// TwinCAT 3 PLC project home
// ProgramVersion: 3.1.4024.0
// libraries:
//   Tc2_Standard, * (Beckhoff Automation GmbH)
//   Tc2_System, * (Beckhoff Automation GmbH)
//   Tc3_Module, * (Beckhoff Automation GmbH)
// project tree:
//   / Food.TcDUT, Fridge.TcDUT, garden.TcPOU, house.TcGVL, Kitchen.TcPOU, main.TcPOU, Plant.TcDUT, Room.TcPOU, task_garden.TcTTO, task_house.TcTTO
// real-time tasks:
//   TASK task_house: cycle T#10ms, priority 20, ADS port 350
//   TASK task_garden: cycle T#10ms, priority 1, ADS port 351

CONFIGURATION home
    RESOURCE PLC ON TwinCAT3
        TASK task_garden(INTERVAL := T#10ms, PRIORITY := 1);
        TASK task_house(INTERVAL := T#10ms, PRIORITY := 20);
        PROGRAM garden WITH task_garden : garden;
        PROGRAM main WITH task_house : main;
    END_RESOURCE
END_CONFIGURATION

// ---- Food.TcDUT
{attribute 'qualified_only'}
{attribute 'strict'}
{attribute 'to_string'}
TYPE Food :
(
    Nothing,
    Carrot,
    Cabbage,
    Broccoli,
    Peas,
    Tofu,
    Humous,
    LentilCurry
);
END_TYPE

// ---- Fridge.TcDUT
TYPE Fridge :
STRUCT
// Store meat at the bottom
    top_shelf    : ARRAY [0..7] OF Food;
    middle_shelf : ARRAY [0..7] OF Food;
    bottom_shelf : ARRAY [0..7] OF Food;
    drawer       : ARRAY [0..3] OF Food;
    door_shelf   : ARRAY [0..3] OF Food;
END_STRUCT
END_TYPE

// ---- Plant.TcDUT
{attribute 'qualified_only'}
{attribute 'strict'}
TYPE Plant :
(
    AppleTree,
    BlackberryBush,
    Grass,
    Ivy,
    Hedge,
    RoseBush
);
END_TYPE

// ---- house.TcGVL
{attribute 'qualified_only'}
VAR_GLOBAL CONSTANT
    ADDRESS     : STRING := '13 Apple Cart Way'; // Next door to 1 Pear Drop Lane
    N_BEDROOMS  : USINT  := 4;
    N_BATHROOMS : USINT  := 1;
END_VAR

// ---- garden.TcPOU
PROGRAM garden
VAR PERSISTENT
    plants                  : ARRAY [0..255] OF Plant;
END_VAR
VAR
    vegetable_plot_at_front : ARRAY [0..4] OF ARRAY [0..2] OF ARRAY [0..7] OF Plant;
    vegetable_plot_at_back  : ARRAY [0..3,0..5,0..6] OF Plant;
END_VAR

END_PROGRAM

// ---- main.TcPOU
PROGRAM main
VAR
    kitchen     : Kitchen;
    dining_room : Room;
    living_room : Room;
    bedroom     : ARRAY [0..(house.N_BEDROOMS-1)]  OF Room;
    bathroom    : ARRAY [0..(house.N_BATHROOMS-1)] OF Room;

    i           : USINT := 0;
END_VAR

kitchen(target_luminosity_lumens := 1300, target_temperature_oc := 19.5, n_broccolis := 3);
dining_room(target_luminosity_lumens := 1100, target_temperature_oc := 19.5);
living_room(target_luminosity_lumens := 800, target_temperature_oc := 19.5);

FOR i := 0 TO (house.N_BEDROOMS-1) DO
    bedroom[i](target_luminosity_lumens := 600, target_temperature_oc := 16.0);
END_FOR

FOR i := 0 TO (house.N_BATHROOMS-1) DO
    bathroom[i](target_luminosity_lumens := 1300, target_temperature_oc := 18.5);
END_FOR

END_PROGRAM

// ---- Kitchen.TcPOU
FUNCTION_BLOCK kitchen EXTENDS room
VAR_INPUT
    n_broccolis : USINT := 0;
END_VAR
VAR PERSISTENT
    fridge      : Fridge;
END_VAR
VAR
    description : STRING := '';
    i           : USINT  := 0;
END_VAR

FOR i := 0 TO MIN(n_broccolis, 7) DO
    fridge.top_shelf[i] := Food.Broccoli;
END_FOR

fridge.middle_shelf[4] := Food.Humous;
fridge.middle_shelf[5] := Food.Tofu;

fridge.bottom_shelf[2] := Food.LentilCurry;

fridge.drawer[0] := Food.Peas;

fridge.door_shelf[0] := Food.Nothing;
fridge.door_shelf[1] := Food.Nothing;
fridge.door_shelf[2] := Food.Nothing;
fridge.door_shelf[3] := Food.Nothing;

description := TO_STRING(fridge.top_shelf[0]);

END_FUNCTION_BLOCK

// ---- Room.TcPOU
FUNCTION_BLOCK room
VAR_INPUT
    target_luminosity_lumens : UINT := 1000;
    target_temperature_oc    : REAL := 18.5;
END_VAR
VAR PERSISTENT
    name                     : STRING;
END_VAR
VAR
    actual_luminosity_lumens : UINT := 1200;
    actual_temperature_oc    : REAL := 18.5;
    is_occupied              : BOOL := FALSE;
    heating_on               : BOOL := FALSE;
END_VAR

heating_on := heating();

METHOD PRIVATE heating : BOOL
VAR_INST
    heating_on                    : BOOL := FALSE;
    was_occupied_at_previous_step : BOOL := FALSE;
    timer                         : TON;
END_VAR
IF is_occupied THEN
    timer(IN := FALSE);
ELSIF was_occupied_at_previous_step AND NOT is_occupied THEN
    timer(
        IN := TRUE,
        PT := TIME#30S,
    );
END_IF

timer();

IF actual_temperature_oc >= target_temperature_oc THEN
    heating_on := FALSE;
ELSIF (actual_temperature_oc < target_temperature_oc) AND is_occupied THEN
    heating_on := TRUE;
ELSIF NOT is_occupied AND timer.Q THEN
    heating_on := FALSE;
END_IF

was_occupied_at_previous_step := is_occupied;

heating := heating_on;
END_METHOD

{attribute 'TcRpcEnable'}
METHOD PRIVATE lights
VAR
    light_on : BOOL := FALSE;
END_VAR
light_on := (actual_luminosity_lumens < target_luminosity_lumens)
         AND is_occupied;
END_METHOD

{attribute 'TcRpcEnable'}
METHOD update_actual_temperature_oc : BOOL
VAR_INPUT
    new_temperature_oc : SINT;
END_VAR
actual_temperature_oc := SINT_TO_REAL(new_temperature_oc);

update_actual_temperature_oc := TRUE;
END_METHOD

END_FUNCTION_BLOCK
